PROGRAM BmsSerialBackground
VAR
	
END_VAR

BMSSerialCtrl(
	Mode:= SERIALLINEMODE_PC_COM_PORT, 
	pComIn:= ADR(pComIn), 
	pComOut:= ADR(pComOut), 
	SizeComIn:= SIZEOF(pComIN), 
	Error=> , 
	ErrorID=> , 
	TxBuffer:= TxBuffer, 
	RxBuffer:= RxBuffer);

END_PROGRAM

(* stored: Version 1.1.0.1, ProductVersion 3.1.4024.14
   POU BmsSerialBackground: Id {4d331f7a-e7eb-479b-8d03-52bcd0d98811}, SpecialFunc None *)
